(* PLC project tri_chain, Dassault Systèmes ControlBuild 2019 FD01 *)
(* stored: creationDateTime 2018-10-05T16:35:32-01:00 *)

CONFIGURATION tri_chain
  VAR_GLOBAL
    cp_trichain/ON AT 5 : BOOL := false;
    cp_trichain/run1 AT 6 : BOOL := false;
    cp_trichain/startSensor1 AT 7 : BOOL := false;
    cp_trichain/endSensor1 AT 8 : BOOL := false;
    cp_trichain/run2 AT 9 : BOOL := false;
    cp_trichain/startSensor2 AT 10 : BOOL := false;
    cp_trichain/endSensor2 AT 11 : BOOL := false;
    cp_trichain/run3 AT 12 : BOOL := false;
    cp_trichain/startSensor3 AT 13 : BOOL := false;
    cp_trichain/endSensor3 AT 14 : BOOL := false;
    cp_trichain/sensor1 AT 15 : BOOL := false;
    cp_trichain/sensor2 AT 16 : BOOL := false;
    cp_trichain/sensor3 AT 17 : BOOL := false;
    cp_trichain/endSensor AT 18 : BOOL := false;
    cp_trichain/endSensor4 AT 19 : BOOL := false;
    cp_trichain/mvt1 AT 20 : BOOL := false;
    cp_trichain/mvt2 AT 21 : BOOL := false;
    cp_trichain/mvt3 AT 22 : BOOL := false;
    cp_trichain/moveToLeft AT 24 : BOOL := false;
    cp_trichain/moveToRight AT 25 : BOOL := false;
    cp_trichain/chainMvt AT 26 : BOOL := false;
    cp_trichain/mvt4 AT 23 : BOOL := false;
    cp_trichain/chain1/globalRunning AT 5 : BOOL := false;
    cp_trichain/chain1/localRunning AT 6 : BOOL := false;
    cp_trichain/chain1/startSensor AT 7 : BOOL := false;
    cp_trichain/chain1/endSensor AT 8 : BOOL := false;
    cp_trichain/chain1/captureEnabled AT 27 : BOOL := false;
    cp_trichain/chain1/movement AT 20 : BOOL := false;
    cp_trichain/chain1/captureRequest AT 30 : BOOL := false;
    cp_trichain/chain1/captureFinished AT 31 : BOOL := false;
    cp_trichain/chain1/_X_10 AT 40 : BOOL := true;
    cp_trichain/chain1/_X_11 AT 41 : BOOL := false;
    cp_trichain/chain1/_X_12 AT 42 : BOOL := false;
    cp_trichain/chain1/_X_13 AT 43 : BOOL := false;
    cp_trichain/chain1/_X_14 AT 44 : BOOL := false;
    cp_trichain/chain1/_X_15 AT 45 : BOOL := false;
    cp_trichain/chain2/globalRunning AT 5 : BOOL := false;
    cp_trichain/chain2/localRunning AT 9 : BOOL := false;
    cp_trichain/chain2/startSensor AT 10 : BOOL := false;
    cp_trichain/chain2/endSensor AT 11 : BOOL := false;
    cp_trichain/chain2/captureEnabled AT 28 : BOOL := false;
    cp_trichain/chain2/movement AT 21 : BOOL := false;
    cp_trichain/chain2/captureRequest AT 32 : BOOL := false;
    cp_trichain/chain2/captureFinished AT 33 : BOOL := false;
    cp_trichain/chain2/_X_10 AT 50 : BOOL := true;
    cp_trichain/chain2/_X_11 AT 51 : BOOL := false;
    cp_trichain/chain2/_X_12 AT 52 : BOOL := false;
    cp_trichain/chain2/_X_13 AT 53 : BOOL := false;
    cp_trichain/chain2/_X_14 AT 54 : BOOL := false;
    cp_trichain/chain2/_X_15 AT 55 : BOOL := false;
    cp_trichain/chain3/globalRunning AT 5 : BOOL := false;
    cp_trichain/chain3/localRunning AT 12 : BOOL := false;
    cp_trichain/chain3/startSensor AT 13 : BOOL := false;
    cp_trichain/chain3/endSensor AT 14 : BOOL := false;
    cp_trichain/chain3/captureEnabled AT 29 : BOOL := false;
    cp_trichain/chain3/movement AT 22 : BOOL := false;
    cp_trichain/chain3/captureRequest AT 34 : BOOL := false;
    cp_trichain/chain3/captureFinished AT 35 : BOOL := false;
    cp_trichain/chain3/_X_10 AT 60 : BOOL := true;
    cp_trichain/chain3/_X_11 AT 61 : BOOL := false;
    cp_trichain/chain3/_X_12 AT 62 : BOOL := false;
    cp_trichain/chain3/_X_13 AT 63 : BOOL := false;
    cp_trichain/chain3/_X_14 AT 64 : BOOL := false;
    cp_trichain/chain3/_X_15 AT 65 : BOOL := false;
    cp_trichain/shuttleControl/globalRunning AT 5 : BOOL := false;
    cp_trichain/shuttleControl/sensorPos1 AT 15 : BOOL := false;
    cp_trichain/shuttleControl/sensorPos2 AT 16 : BOOL := false;
    cp_trichain/shuttleControl/sensorPos3 AT 17 : BOOL := false;
    cp_trichain/shuttleControl/requestCapture1 AT 30 : BOOL := false;
    cp_trichain/shuttleControl/endCapture1 AT 31 : BOOL := false;
    cp_trichain/shuttleControl/requestCapture2 AT 32 : BOOL := false;
    cp_trichain/shuttleControl/endCapture2 AT 33 : BOOL := false;
    cp_trichain/shuttleControl/requestCapture3 AT 34 : BOOL := false;
    cp_trichain/shuttleControl/endCapture3 AT 35 : BOOL := false;
    cp_trichain/shuttleControl/depositRequest AT 36 : BOOL := false;
    cp_trichain/shuttleControl/depositFinished AT 37 : BOOL := false;
    cp_trichain/shuttleControl/enableCapture1 AT 27 : BOOL := false;
    cp_trichain/shuttleControl/enableCapture2 AT 28 : BOOL := false;
    cp_trichain/shuttleControl/enableCapture3 AT 29 : BOOL := false;
    cp_trichain/shuttleControl/enableCapture AT 39 : BOOL := false;
    cp_trichain/shuttleControl/enableDeposit AT 38 : BOOL := false;
    cp_trichain/shuttleControl/moveToLeft AT 24 : BOOL := false;
    cp_trichain/shuttleControl/moveToRight AT 25 : BOOL := false;
    cp_trichain/shuttleControl/goTo1 AT 70 : BOOL := false;
    cp_trichain/shuttleControl/goTo2 AT 71 : BOOL := false;
    cp_trichain/shuttleControl/goTo3 AT 72 : BOOL := false;
    cp_trichain/shuttleControl/shuttleInPosition AT 73 : BOOL := false;
    cp_trichain/shuttleControl/_X_10 AT 74 : BOOL := true;
    cp_trichain/shuttleControl/_X_15 AT 82 : BOOL := false;
    cp_trichain/shuttleControl/_X_13 AT 80 : BOOL := false;
    cp_trichain/shuttleControl/_X_11 AT 75 : BOOL := false;
    cp_trichain/shuttleControl/_X_16 AT 83 : BOOL := false;
    cp_trichain/shuttleControl/_X_14 AT 81 : BOOL := false;
    cp_trichain/shuttleControl/_X_12 AT 76 : BOOL := false;
    cp_trichain/shuttleControl/_X_17 AT 77 : BOOL := false;
    cp_trichain/shuttleControl/_X_18 AT 78 : BOOL := false;
    cp_trichain/shuttleControl/_X_19 AT 79 : BOOL := false;
    cp_trichain/shuttleControl/_X_20 AT 84 : BOOL := true;
    cp_trichain/shuttleControl/_X_21 AT 85 : BOOL := false;
    cp_trichain/shuttleControl/_X_22 AT 86 : BOOL := false;
    cp_trichain/shuttleControl/_X_30 AT 87 : BOOL := true;
    cp_trichain/shuttleControl/_X_31 AT 88 : BOOL := false;
    cp_trichain/shuttleControl/_X_32 AT 89 : BOOL := false;
    cp_trichain/shuttleControl/_X_40 AT 90 : BOOL := true;
    cp_trichain/shuttleControl/_X_41 AT 91 : BOOL := false;
    cp_trichain/shuttleControl/_X_42 AT 92 : BOOL := false;
    cp_trichain/shuttleChain/globalRunning AT 5 : BOOL := false;
    cp_trichain/shuttleChain/endSensor AT 18 : BOOL := false;
    cp_trichain/shuttleChain/depositEnabled AT 38 : BOOL := false;
    cp_trichain/shuttleChain/captureEnabled AT 39 : BOOL := false;
    cp_trichain/shuttleChain/movement AT 26 : BOOL := false;
    cp_trichain/shuttleChain/depositRequest AT 36 : BOOL := false;
    cp_trichain/shuttleChain/depositFinished AT 37 : BOOL := false;
    cp_trichain/shuttleChain/_X_10 AT 108 : BOOL := true;
    cp_trichain/shuttleChain/_X_11 AT 109 : BOOL := false;
    cp_trichain/shuttleChain/_X_12 AT 110 : BOOL := false;
    cp_trichain/shuttleChain/_X_13 AT 111 : BOOL := false;
    cp_trichain/shuttleChain/_X_14 AT 112 : BOOL := false;
    cp_trichain/outputChain/globalRunning AT 5 : BOOL := false;
    cp_trichain/outputChain/depositEnabled AT 38 : BOOL := false;
    cp_trichain/outputChain/endSensor AT 19 : BOOL := false;
    cp_trichain/outputChain/movement AT 23 : BOOL := false;
    cp_trichain/outputChain/_X_10 AT 117 : BOOL := true;
    cp_trichain/outputChain/_X_11 AT 118 : BOOL := false;
    cp_trichain/outputChain/_X_12 AT 119 : BOOL := false;
    op_trichain/mvt1 AT 20 : BOOL := false;
    op_trichain/mvt2 AT 21 : BOOL := false;
    op_trichain/mvt3 AT 22 : BOOL := false;
    op_trichain/mvt4 AT 23 : BOOL := false;
    op_trichain/moveToLeft AT 24 : BOOL := false;
    op_trichain/moveToRight AT 25 : BOOL := false;
    op_trichain/chainMvt AT 26 : BOOL := false;
    op_trichain/ON AT 5 : BOOL := false;
    op_trichain/run1 AT 6 : BOOL := false;
    op_trichain/startSensor1 AT 7 : BOOL := false;
    op_trichain/endSensor1 AT 8 : BOOL := false;
    op_trichain/run2 AT 9 : BOOL := false;
    op_trichain/startSensor2 AT 10 : BOOL := false;
    op_trichain/endSensor2 AT 11 : BOOL := false;
    op_trichain/run3 AT 12 : BOOL := false;
    op_trichain/startSensor3 AT 13 : BOOL := false;
    op_trichain/endSensor3 AT 14 : BOOL := false;
    op_trichain/endSensor4 AT 19 : BOOL := false;
    op_trichain/sensor1 AT 15 : BOOL := false;
    op_trichain/sensor2 AT 16 : BOOL := false;
    op_trichain/sensor3 AT 17 : BOOL := false;
    op_trichain/endSensor AT 18 : BOOL := false;
    op_trichain/creation1/idProd AT 525 : DINT := 0;
    op_trichain/creation1/creationFailed AT 126 : BOOL := false;
    op_trichain/creation1/status_act_prod AT 526 : DINT := 0;
    op_trichain/creation1/m11 AT 17 : REAL := 1502.68;
    op_trichain/creation1/m12 AT 18 : REAL := 0.0;
    op_trichain/creation1/m13 AT 19 : REAL := -2.44921e-014;
    op_trichain/creation1/m14 AT 20 : REAL := 5480.36;
    op_trichain/creation1/m21 AT 21 : REAL := 0.0;
    op_trichain/creation1/m22 AT 22 : REAL := 2997.32;
    op_trichain/creation1/m23 AT 23 : REAL := 0.0;
    op_trichain/creation1/m24 AT 24 : REAL := 27006.2;
    op_trichain/creation1/m31 AT 25 : REAL := 3.68038e-013;
    op_trichain/creation1/m32 AT 26 : REAL := 0.0;
    op_trichain/creation1/m33 AT 27 : REAL := 100.0;
    op_trichain/creation1/m34 AT 28 : REAL := 1.0;
    op_trichain/creation1/m41 AT 29 : REAL := 0.0;
    op_trichain/creation1/m42 AT 30 : REAL := 0.0;
    op_trichain/creation1/m43 AT 31 : REAL := 0.0;
    op_trichain/creation1/m44 AT 32 : REAL := 1.0;
    op_trichain/creation1/px AT 33 : REAL := 5600.0;
    op_trichain/creation1/py AT 34 : REAL := 27000.0;
    op_trichain/creation1/pz AT 35 : REAL := 1.5;
    op_trichain/creation1/dx AT 36 : REAL := 1500.0;
    op_trichain/creation1/dy AT 37 : REAL := 3000.0;
    op_trichain/creation1/dz AT 38 : REAL := 100.0;
    op_trichain/creation1/presenceProduct AT 127 : BOOL := false;
    op_trichain/creation1/arrival_PB AT 128 : BOOL := false;
    op_trichain/creation1/time2reach AT 39 : REAL := 0.0;
    op_trichain/creation1/edge_arrival_PB AT 129 : BOOL := false;
    op_trichain/creation1/first AT 130 : BOOL := true;
    op_trichain/creation1/pulseType AT 131 : BOOL := true;
    op_trichain/creation1/pulseDuration AT 40 : REAL := 10.0;
    op_trichain/chain1/forward AT 20 : BOOL := false;
    op_trichain/chain1/localRun AT 6 : BOOL := false;
    op_trichain/chain1/start_sensor AT 7 : BOOL := false;
    op_trichain/chain1/end_sensor AT 8 : BOOL := false;
    op_trichain/chain1/motor1dir/forward AT 20 : BOOL := false;
    op_trichain/chain1/motor1dir/cmdSupply AT 138 : BOOL := true;
    op_trichain/chain1/motor1dir/sensorSupply AT 137 : BOOL := true;
    op_trichain/chain1/motor1dir/voltage380 AT 136 : BOOL := true;
    op_trichain/chain1/motor1dir/speedVal AT 42 : REAL := 0.0;
    op_trichain/chain1/motor1dir/speedPercent AT 41 : REAL := 0.0;
    op_trichain/chain1/motor1dir/thermal AT 135 : BOOL := false;
    op_trichain/chain1/motor1dir/forwardFB AT 134 : BOOL := false;
    op_trichain/chain1/motor1dir/increment AT 43 : REAL := 0.0;
    op_trichain/chain1/motor1dir/memoFwd AT 139 : BOOL := false;
    op_trichain/chain1/motor1dir/forwardState AT 140 : BOOL := false;
    op_trichain/chain1/motor1dir/wantedSpeed AT 44 : REAL := 0.0;
    op_trichain/chain1/motor1dir/nominalSpeed AT 45 : REAL := 500.0;
    op_trichain/chain1/motor1dir/nominalTime AT 46 : REAL := 0.1;
    op_trichain/chain1/motor1dir/thermalLogic AT 141 : BOOL := false;
    op_trichain/chain1/motor1dir/feedbackLogic AT 142 : BOOL := true;
    op_trichain/chain1/motor1dir/d_locking AT 143 : BOOL := false;
    op_trichain/chain1/motor1dir/v_d_locking AT 47 : REAL := 0.0;
    op_trichain/chain1/motor1dir/d_feedback AT 144 : BOOL := false;
    op_trichain/chain1/motor1dir/v_d_feedback AT 145 : BOOL := false;
    op_trichain/chain1/motor1dir/d_electrical AT 146 : BOOL := false;
    op_trichain/chain1/motor1dir/v_d_electrical AT 147 : BOOL := false;
    op_trichain/chain1/runButton/output AT 6 : BOOL := false;
    op_trichain/chain1/runButton/user_PushButton AT 148 : BOOL := false;
    op_trichain/chain1/runButton/time2reach AT 149 : BOOL := false;
    op_trichain/chain1/runButton/pulse_type AT 150 : BOOL := false;
    op_trichain/chain1/runButton/pulseDuration AT 48 : REAL := 2.0;
    op_trichain/chain1/start_sensor/sensorSupply AT 133 : BOOL := true;
    op_trichain/chain1/start_sensor/passing AT 7 : BOOL := false;
    op_trichain/chain1/start_sensor/status_act_prod AT 527 : DINT := 0;
    op_trichain/chain1/start_sensor/m11 AT 49 : REAL := 498.214;
    op_trichain/chain1/start_sensor/m12 AT 50 : REAL := 0.0;
    op_trichain/chain1/start_sensor/m13 AT 51 : REAL := -2.44921e-014;
    op_trichain/chain1/start_sensor/m14 AT 52 : REAL := 5223.22;
    op_trichain/chain1/start_sensor/m21 AT 53 : REAL := 0.0;
    op_trichain/chain1/start_sensor/m22 AT 54 : REAL := 498.214;
    op_trichain/chain1/start_sensor/m23 AT 55 : REAL := 0.0;
    op_trichain/chain1/start_sensor/m24 AT 56 : REAL := 26998.2;
    op_trichain/chain1/start_sensor/m31 AT 57 : REAL := 1.22023e-013;
    op_trichain/chain1/start_sensor/m32 AT 58 : REAL := 0.0;
    op_trichain/chain1/start_sensor/m33 AT 59 : REAL := 100.0;
    op_trichain/chain1/start_sensor/m34 AT 60 : REAL := 1.0;
    op_trichain/chain1/start_sensor/m41 AT 61 : REAL := 0.0;
    op_trichain/chain1/start_sensor/m42 AT 62 : REAL := 0.0;
    op_trichain/chain1/start_sensor/m43 AT 63 : REAL := 0.0;
    op_trichain/chain1/start_sensor/m44 AT 64 : REAL := 1.0;
    op_trichain/chain1/start_sensor/px AT 65 : REAL := 4500.0;
    op_trichain/chain1/start_sensor/py AT 66 : REAL := 27000.0;
    op_trichain/chain1/start_sensor/pz AT 67 : REAL := 0.0;
    op_trichain/chain1/start_sensor/dx AT 68 : REAL := 500.0;
    op_trichain/chain1/start_sensor/dy AT 69 : REAL := 500.0;
    op_trichain/chain1/start_sensor/dz AT 70 : REAL := 100.0;
    op_trichain/chain1/start_sensor/detection AT 151 : BOOL := false;
    op_trichain/chain1/start_sensor/passingLogic AT 152 : BOOL := true;
    op_trichain/chain1/start_sensor/d_passing AT 153 : BOOL := false;
    op_trichain/chain1/start_sensor/v_d_passing AT 154 : BOOL := true;
    op_trichain/chain1/end_sensor/sensorSupply AT 132 : BOOL := true;
    op_trichain/chain1/end_sensor/passing AT 8 : BOOL := false;
    op_trichain/chain1/end_sensor/status_act_prod AT 528 : DINT := 0;
    op_trichain/chain1/end_sensor/m11 AT 71 : REAL := 498.214;
    op_trichain/chain1/end_sensor/m12 AT 72 : REAL := 0.0;
    op_trichain/chain1/end_sensor/m13 AT 73 : REAL := -2.44921e-014;
    op_trichain/chain1/end_sensor/m14 AT 74 : REAL := 3334.82;
    op_trichain/chain1/end_sensor/m21 AT 75 : REAL := 0.0;
    op_trichain/chain1/end_sensor/m22 AT 76 : REAL := 498.214;
    op_trichain/chain1/end_sensor/m23 AT 77 : REAL := 0.0;
    op_trichain/chain1/end_sensor/m24 AT 78 : REAL := 19999.1;
    op_trichain/chain1/end_sensor/m31 AT 79 : REAL := 1.22023e-013;
    op_trichain/chain1/end_sensor/m32 AT 80 : REAL := 0.0;
    op_trichain/chain1/end_sensor/m33 AT 81 : REAL := 100.0;
    op_trichain/chain1/end_sensor/m34 AT 82 : REAL := 1.05;
    op_trichain/chain1/end_sensor/m41 AT 83 : REAL := 0.0;
    op_trichain/chain1/end_sensor/m42 AT 84 : REAL := 0.0;
    op_trichain/chain1/end_sensor/m43 AT 85 : REAL := 0.0;
    op_trichain/chain1/end_sensor/m44 AT 86 : REAL := 1.0;
    op_trichain/chain1/end_sensor/px AT 87 : REAL := 2850.0;
    op_trichain/chain1/end_sensor/py AT 88 : REAL := 20000.0;
    op_trichain/chain1/end_sensor/pz AT 89 : REAL := 0.0;
    op_trichain/chain1/end_sensor/dx AT 90 : REAL := 500.0;
    op_trichain/chain1/end_sensor/dy AT 91 : REAL := 500.0;
    op_trichain/chain1/end_sensor/dz AT 92 : REAL := 100.0;
    op_trichain/chain1/end_sensor/detection AT 155 : BOOL := false;
    op_trichain/chain1/end_sensor/passingLogic AT 156 : BOOL := true;
    op_trichain/chain1/end_sensor/d_passing AT 157 : BOOL := false;
    op_trichain/chain1/end_sensor/v_d_passing AT 158 : BOOL := true;
    op_trichain/chain1/chain/linearSpeed AT 42 : REAL := 0.0;
    op_trichain/chain1/chain/status_act_prod AT 529 : DINT := 0;
    op_trichain/chain1/chain/m11 AT 93 : REAL := 4001.79;
    op_trichain/chain1/chain/m12 AT 94 : REAL := 0.0;
    op_trichain/chain1/chain/m13 AT 95 : REAL := -2.44921e-014;
    op_trichain/chain1/chain/m14 AT 96 : REAL := 2981.25;
    op_trichain/chain1/chain/m21 AT 97 : REAL := 0.0;
    op_trichain/chain1/chain/m22 AT 98 : REAL := 9996.43;
    op_trichain/chain1/chain/m23 AT 99 : REAL := 0.0;
    op_trichain/chain1/chain/m24 AT 100 : REAL := 18102.7;
    op_trichain/chain1/chain/m31 AT 101 : REAL := 9.80123e-013;
    op_trichain/chain1/chain/m32 AT 102 : REAL := 0.0;
    op_trichain/chain1/chain/m33 AT 103 : REAL := 100.0;
    op_trichain/chain1/chain/m34 AT 104 : REAL := 1.0;
    op_trichain/chain1/chain/m41 AT 105 : REAL := 0.0;
    op_trichain/chain1/chain/m42 AT 106 : REAL := 0.0;
    op_trichain/chain1/chain/m43 AT 107 : REAL := 0.0;
    op_trichain/chain1/chain/m44 AT 108 : REAL := 1.0;
    op_trichain/chain1/chain/px AT 109 : REAL := 2500.0;
    op_trichain/chain1/chain/py AT 110 : REAL := 18100.0;
    op_trichain/chain1/chain/pz AT 111 : REAL := 1.0;
    op_trichain/chain1/chain/dx AT 112 : REAL := 4000.0;
    op_trichain/chain1/chain/dy AT 113 : REAL := 10000.0;
    op_trichain/chain1/chain/dz AT 114 : REAL := 100.0;
    op_trichain/chain1/chain/sProduct AT 115 : REAL := 0.0;
    op_trichain/chain1/chain/interaction AT 159 : BOOL := false;
    op_trichain/chain1/chain/d_locking AT 160 : BOOL := false;
    op_trichain/chain1/chain/v_d_locking AT 161 : BOOL := false;
    op_trichain/chain2/forward AT 21 : BOOL := false;
    op_trichain/chain2/localRun AT 9 : BOOL := false;
    op_trichain/chain2/start_sensor AT 10 : BOOL := false;
    op_trichain/chain2/end_sensor AT 11 : BOOL := false;
    op_trichain/chain2/motor1dir/forward AT 21 : BOOL := false;
    op_trichain/chain2/motor1dir/cmdSupply AT 168 : BOOL := true;
    op_trichain/chain2/motor1dir/sensorSupply AT 167 : BOOL := true;
    op_trichain/chain2/motor1dir/voltage380 AT 166 : BOOL := true;
    op_trichain/chain2/motor1dir/speedVal AT 117 : REAL := 0.0;
    op_trichain/chain2/motor1dir/speedPercent AT 116 : REAL := 0.0;
    op_trichain/chain2/motor1dir/thermal AT 165 : BOOL := false;
    op_trichain/chain2/motor1dir/forwardFB AT 164 : BOOL := false;
    op_trichain/chain2/motor1dir/increment AT 118 : REAL := 0.0;
    op_trichain/chain2/motor1dir/memoFwd AT 169 : BOOL := false;
    op_trichain/chain2/motor1dir/forwardState AT 170 : BOOL := false;
    op_trichain/chain2/motor1dir/wantedSpeed AT 119 : REAL := 0.0;
    op_trichain/chain2/motor1dir/nominalSpeed AT 120 : REAL := 500.0;
    op_trichain/chain2/motor1dir/nominalTime AT 121 : REAL := 0.1;
    op_trichain/chain2/motor1dir/thermalLogic AT 171 : BOOL := false;
    op_trichain/chain2/motor1dir/feedbackLogic AT 172 : BOOL := true;
    op_trichain/chain2/motor1dir/d_locking AT 173 : BOOL := false;
    op_trichain/chain2/motor1dir/v_d_locking AT 122 : REAL := 0.0;
    op_trichain/chain2/motor1dir/d_feedback AT 174 : BOOL := false;
    op_trichain/chain2/motor1dir/v_d_feedback AT 175 : BOOL := false;
    op_trichain/chain2/motor1dir/d_electrical AT 176 : BOOL := false;
    op_trichain/chain2/motor1dir/v_d_electrical AT 177 : BOOL := false;
    op_trichain/chain2/runButton/output AT 9 : BOOL := false;
    op_trichain/chain2/runButton/user_PushButton AT 178 : BOOL := false;
    op_trichain/chain2/runButton/time2reach AT 179 : BOOL := false;
    op_trichain/chain2/runButton/pulse_type AT 180 : BOOL := false;
    op_trichain/chain2/runButton/pulseDuration AT 123 : REAL := 2.0;
    op_trichain/chain2/start_sensor/sensorSupply AT 163 : BOOL := true;
    op_trichain/chain2/start_sensor/passing AT 10 : BOOL := false;
    op_trichain/chain2/start_sensor/status_act_prod AT 530 : DINT := 0;
    op_trichain/chain2/start_sensor/m11 AT 124 : REAL := 500.0;
    op_trichain/chain2/start_sensor/m12 AT 125 : REAL := 0.0;
    op_trichain/chain2/start_sensor/m13 AT 126 : REAL := 0.0;
    op_trichain/chain2/start_sensor/m14 AT 127 : REAL := 8500.0;
    op_trichain/chain2/start_sensor/m21 AT 128 : REAL := 0.0;
    op_trichain/chain2/start_sensor/m22 AT 129 : REAL := 500.0;
    op_trichain/chain2/start_sensor/m23 AT 130 : REAL := 0.0;
    op_trichain/chain2/start_sensor/m24 AT 131 : REAL := 27000.0;
    op_trichain/chain2/start_sensor/m31 AT 132 : REAL := 0.0;
    op_trichain/chain2/start_sensor/m32 AT 133 : REAL := 0.0;
    op_trichain/chain2/start_sensor/m33 AT 134 : REAL := 100.0;
    op_trichain/chain2/start_sensor/m34 AT 135 : REAL := 0.0;
    op_trichain/chain2/start_sensor/m41 AT 136 : REAL := 0.0;
    op_trichain/chain2/start_sensor/m42 AT 137 : REAL := 0.0;
    op_trichain/chain2/start_sensor/m43 AT 138 : REAL := 0.0;
    op_trichain/chain2/start_sensor/m44 AT 139 : REAL := 1.0;
    op_trichain/chain2/start_sensor/px AT 140 : REAL := 8500.0;
    op_trichain/chain2/start_sensor/py AT 141 : REAL := 27000.0;
    op_trichain/chain2/start_sensor/pz AT 142 : REAL := 0.0;
    op_trichain/chain2/start_sensor/dx AT 143 : REAL := 500.0;
    op_trichain/chain2/start_sensor/dy AT 144 : REAL := 500.0;
    op_trichain/chain2/start_sensor/dz AT 145 : REAL := 100.0;
    op_trichain/chain2/start_sensor/detection AT 181 : BOOL := false;
    op_trichain/chain2/start_sensor/passingLogic AT 182 : BOOL := true;
    op_trichain/chain2/start_sensor/d_passing AT 183 : BOOL := false;
    op_trichain/chain2/start_sensor/v_d_passing AT 184 : BOOL := true;
    op_trichain/chain2/end_sensor/sensorSupply AT 162 : BOOL := true;
    op_trichain/chain2/end_sensor/passing AT 11 : BOOL := false;
    op_trichain/chain2/end_sensor/status_act_prod AT 531 : DINT := 0;
    op_trichain/chain2/end_sensor/m11 AT 146 : REAL := 500.0;
    op_trichain/chain2/end_sensor/m12 AT 147 : REAL := 0.0;
    op_trichain/chain2/end_sensor/m13 AT 148 : REAL := 0.0;
    op_trichain/chain2/end_sensor/m14 AT 149 : REAL := 6900.0;
    op_trichain/chain2/end_sensor/m21 AT 150 : REAL := 0.0;
    op_trichain/chain2/end_sensor/m22 AT 151 : REAL := 500.0;
    op_trichain/chain2/end_sensor/m23 AT 152 : REAL := 0.0;
    op_trichain/chain2/end_sensor/m24 AT 153 : REAL := 20000.0;
    op_trichain/chain2/end_sensor/m31 AT 154 : REAL := 0.0;
    op_trichain/chain2/end_sensor/m32 AT 155 : REAL := 0.0;
    op_trichain/chain2/end_sensor/m33 AT 156 : REAL := 100.0;
    op_trichain/chain2/end_sensor/m34 AT 157 : REAL := 0.0;
    op_trichain/chain2/end_sensor/m41 AT 158 : REAL := 0.0;
    op_trichain/chain2/end_sensor/m42 AT 159 : REAL := 0.0;
    op_trichain/chain2/end_sensor/m43 AT 160 : REAL := 0.0;
    op_trichain/chain2/end_sensor/m44 AT 161 : REAL := 1.0;
    op_trichain/chain2/end_sensor/px AT 162 : REAL := 6900.0;
    op_trichain/chain2/end_sensor/py AT 163 : REAL := 20000.0;
    op_trichain/chain2/end_sensor/pz AT 164 : REAL := 0.0;
    op_trichain/chain2/end_sensor/dx AT 165 : REAL := 500.0;
    op_trichain/chain2/end_sensor/dy AT 166 : REAL := 500.0;
    op_trichain/chain2/end_sensor/dz AT 167 : REAL := 100.0;
    op_trichain/chain2/end_sensor/detection AT 185 : BOOL := false;
    op_trichain/chain2/end_sensor/passingLogic AT 186 : BOOL := true;
    op_trichain/chain2/end_sensor/d_passing AT 187 : BOOL := false;
    op_trichain/chain2/end_sensor/v_d_passing AT 188 : BOOL := true;
    op_trichain/chain2/chain/linearSpeed AT 117 : REAL := 0.0;
    op_trichain/chain2/chain/status_act_prod AT 532 : DINT := 0;
    op_trichain/chain2/chain/m11 AT 168 : REAL := 4000.0;
    op_trichain/chain2/chain/m12 AT 169 : REAL := 0.0;
    op_trichain/chain2/chain/m13 AT 170 : REAL := 0.0;
    op_trichain/chain2/chain/m14 AT 171 : REAL := 6500.0;
    op_trichain/chain2/chain/m21 AT 172 : REAL := 0.0;
    op_trichain/chain2/chain/m22 AT 173 : REAL := 10000.0;
    op_trichain/chain2/chain/m23 AT 174 : REAL := 0.0;
    op_trichain/chain2/chain/m24 AT 175 : REAL := 18100.0;
    op_trichain/chain2/chain/m31 AT 176 : REAL := 0.0;
    op_trichain/chain2/chain/m32 AT 177 : REAL := 0.0;
    op_trichain/chain2/chain/m33 AT 178 : REAL := 100.0;
    op_trichain/chain2/chain/m34 AT 179 : REAL := 0.0;
    op_trichain/chain2/chain/m41 AT 180 : REAL := 0.0;
    op_trichain/chain2/chain/m42 AT 181 : REAL := 0.0;
    op_trichain/chain2/chain/m43 AT 182 : REAL := 0.0;
    op_trichain/chain2/chain/m44 AT 183 : REAL := 1.0;
    op_trichain/chain2/chain/px AT 184 : REAL := 6500.0;
    op_trichain/chain2/chain/py AT 185 : REAL := 18100.0;
    op_trichain/chain2/chain/pz AT 186 : REAL := 0.0;
    op_trichain/chain2/chain/dx AT 187 : REAL := 4000.0;
    op_trichain/chain2/chain/dy AT 188 : REAL := 10000.0;
    op_trichain/chain2/chain/dz AT 189 : REAL := 100.0;
    op_trichain/chain2/chain/sProduct AT 190 : REAL := 0.0;
    op_trichain/chain2/chain/interaction AT 189 : BOOL := false;
    op_trichain/chain2/chain/d_locking AT 190 : BOOL := false;
    op_trichain/chain2/chain/v_d_locking AT 191 : BOOL := false;
    op_trichain/creation2/idProd AT 524 : DINT := 0;
    op_trichain/creation2/creationFailed AT 125 : BOOL := false;
    op_trichain/creation2/status_act_prod AT 533 : DINT := 0;
    op_trichain/creation2/m11 AT 191 : REAL := 1500.0;
    op_trichain/creation2/m12 AT 192 : REAL := 0.0;
    op_trichain/creation2/m13 AT 193 : REAL := 0.0;
    op_trichain/creation2/m14 AT 194 : REAL := 9000.0;
    op_trichain/creation2/m21 AT 195 : REAL := 0.0;
    op_trichain/creation2/m22 AT 196 : REAL := 3000.0;
    op_trichain/creation2/m23 AT 197 : REAL := 0.0;
    op_trichain/creation2/m24 AT 198 : REAL := 27000.0;
    op_trichain/creation2/m31 AT 199 : REAL := 0.0;
    op_trichain/creation2/m32 AT 200 : REAL := 0.0;
    op_trichain/creation2/m33 AT 201 : REAL := 100.0;
    op_trichain/creation2/m34 AT 202 : REAL := 0.0;
    op_trichain/creation2/m41 AT 203 : REAL := 0.0;
    op_trichain/creation2/m42 AT 204 : REAL := 0.0;
    op_trichain/creation2/m43 AT 205 : REAL := 0.0;
    op_trichain/creation2/m44 AT 206 : REAL := 1.0;
    op_trichain/creation2/px AT 207 : REAL := 8990.0;
    op_trichain/creation2/py AT 208 : REAL := 27000.0;
    op_trichain/creation2/pz AT 209 : REAL := 1.5;
    op_trichain/creation2/dx AT 210 : REAL := 1500.0;
    op_trichain/creation2/dy AT 211 : REAL := 3000.0;
    op_trichain/creation2/dz AT 212 : REAL := 100.0;
    op_trichain/creation2/presenceProduct AT 192 : BOOL := false;
    op_trichain/creation2/arrival_PB AT 193 : BOOL := false;
    op_trichain/creation2/time2reach AT 213 : REAL := 0.0;
    op_trichain/creation2/edge_arrival_PB AT 194 : BOOL := false;
    op_trichain/creation2/first AT 195 : BOOL := true;
    op_trichain/creation2/pulseType AT 196 : BOOL := true;
    op_trichain/creation2/pulseDuration AT 214 : REAL := 10.0;
    op_trichain/chain3/forward AT 22 : BOOL := false;
    op_trichain/chain3/localRun AT 12 : BOOL := false;
    op_trichain/chain3/start_sensor AT 13 : BOOL := false;
    op_trichain/chain3/end_sensor AT 14 : BOOL := false;
    op_trichain/chain3/motor1dir/forward AT 22 : BOOL := false;
    op_trichain/chain3/motor1dir/cmdSupply AT 203 : BOOL := true;
    op_trichain/chain3/motor1dir/sensorSupply AT 202 : BOOL := true;
    op_trichain/chain3/motor1dir/voltage380 AT 201 : BOOL := true;
    op_trichain/chain3/motor1dir/speedVal AT 216 : REAL := 0.0;
    op_trichain/chain3/motor1dir/speedPercent AT 215 : REAL := 0.0;
    op_trichain/chain3/motor1dir/thermal AT 200 : BOOL := false;
    op_trichain/chain3/motor1dir/forwardFB AT 199 : BOOL := false;
    op_trichain/chain3/motor1dir/increment AT 217 : REAL := 0.0;
    op_trichain/chain3/motor1dir/memoFwd AT 204 : BOOL := false;
    op_trichain/chain3/motor1dir/forwardState AT 205 : BOOL := false;
    op_trichain/chain3/motor1dir/wantedSpeed AT 218 : REAL := 0.0;
    op_trichain/chain3/motor1dir/nominalSpeed AT 219 : REAL := 500.0;
    op_trichain/chain3/motor1dir/nominalTime AT 220 : REAL := 0.1;
    op_trichain/chain3/motor1dir/thermalLogic AT 206 : BOOL := false;
    op_trichain/chain3/motor1dir/feedbackLogic AT 207 : BOOL := true;
    op_trichain/chain3/motor1dir/d_locking AT 208 : BOOL := false;
    op_trichain/chain3/motor1dir/v_d_locking AT 221 : REAL := 0.0;
    op_trichain/chain3/motor1dir/d_feedback AT 209 : BOOL := false;
    op_trichain/chain3/motor1dir/v_d_feedback AT 210 : BOOL := false;
    op_trichain/chain3/motor1dir/d_electrical AT 211 : BOOL := false;
    op_trichain/chain3/motor1dir/v_d_electrical AT 212 : BOOL := false;
    op_trichain/chain3/runButton/output AT 12 : BOOL := false;
    op_trichain/chain3/runButton/user_PushButton AT 213 : BOOL := false;
    op_trichain/chain3/runButton/time2reach AT 214 : BOOL := false;
    op_trichain/chain3/runButton/pulse_type AT 215 : BOOL := false;
    op_trichain/chain3/runButton/pulseDuration AT 222 : REAL := 2.0;
    op_trichain/chain3/start_sensor/sensorSupply AT 198 : BOOL := true;
    op_trichain/chain3/start_sensor/passing AT 13 : BOOL := false;
    op_trichain/chain3/start_sensor/status_act_prod AT 534 : DINT := 0;
    op_trichain/chain3/start_sensor/m11 AT 223 : REAL := 500.0;
    op_trichain/chain3/start_sensor/m12 AT 224 : REAL := 0.0;
    op_trichain/chain3/start_sensor/m13 AT 225 : REAL := 0.0;
    op_trichain/chain3/start_sensor/m14 AT 226 : REAL := 12500.0;
    op_trichain/chain3/start_sensor/m21 AT 227 : REAL := 0.0;
    op_trichain/chain3/start_sensor/m22 AT 228 : REAL := 500.0;
    op_trichain/chain3/start_sensor/m23 AT 229 : REAL := 0.0;
    op_trichain/chain3/start_sensor/m24 AT 230 : REAL := 27000.0;
    op_trichain/chain3/start_sensor/m31 AT 231 : REAL := 0.0;
    op_trichain/chain3/start_sensor/m32 AT 232 : REAL := 0.0;
    op_trichain/chain3/start_sensor/m33 AT 233 : REAL := 100.0;
    op_trichain/chain3/start_sensor/m34 AT 234 : REAL := 0.0;
    op_trichain/chain3/start_sensor/m41 AT 235 : REAL := 0.0;
    op_trichain/chain3/start_sensor/m42 AT 236 : REAL := 0.0;
    op_trichain/chain3/start_sensor/m43 AT 237 : REAL := 0.0;
    op_trichain/chain3/start_sensor/m44 AT 238 : REAL := 1.0;
    op_trichain/chain3/start_sensor/px AT 239 : REAL := 12500.0;
    op_trichain/chain3/start_sensor/py AT 240 : REAL := 27000.0;
    op_trichain/chain3/start_sensor/pz AT 241 : REAL := 0.0;
    op_trichain/chain3/start_sensor/dx AT 242 : REAL := 500.0;
    op_trichain/chain3/start_sensor/dy AT 243 : REAL := 500.0;
    op_trichain/chain3/start_sensor/dz AT 244 : REAL := 100.0;
    op_trichain/chain3/start_sensor/detection AT 216 : BOOL := false;
    op_trichain/chain3/start_sensor/passingLogic AT 217 : BOOL := true;
    op_trichain/chain3/start_sensor/d_passing AT 218 : BOOL := false;
    op_trichain/chain3/start_sensor/v_d_passing AT 219 : BOOL := true;
    op_trichain/chain3/end_sensor/sensorSupply AT 197 : BOOL := true;
    op_trichain/chain3/end_sensor/passing AT 14 : BOOL := false;
    op_trichain/chain3/end_sensor/status_act_prod AT 535 : DINT := 0;
    op_trichain/chain3/end_sensor/m11 AT 245 : REAL := 500.0;
    op_trichain/chain3/end_sensor/m12 AT 246 : REAL := 0.0;
    op_trichain/chain3/end_sensor/m13 AT 247 : REAL := 0.0;
    op_trichain/chain3/end_sensor/m14 AT 248 : REAL := 10950.0;
    op_trichain/chain3/end_sensor/m21 AT 249 : REAL := 0.0;
    op_trichain/chain3/end_sensor/m22 AT 250 : REAL := 500.0;
    op_trichain/chain3/end_sensor/m23 AT 251 : REAL := 0.0;
    op_trichain/chain3/end_sensor/m24 AT 252 : REAL := 20000.0;
    op_trichain/chain3/end_sensor/m31 AT 253 : REAL := 0.0;
    op_trichain/chain3/end_sensor/m32 AT 254 : REAL := 0.0;
    op_trichain/chain3/end_sensor/m33 AT 255 : REAL := 100.0;
    op_trichain/chain3/end_sensor/m34 AT 256 : REAL := 0.0;
    op_trichain/chain3/end_sensor/m41 AT 257 : REAL := 0.0;
    op_trichain/chain3/end_sensor/m42 AT 258 : REAL := 0.0;
    op_trichain/chain3/end_sensor/m43 AT 259 : REAL := 0.0;
    op_trichain/chain3/end_sensor/m44 AT 260 : REAL := 1.0;
    op_trichain/chain3/end_sensor/px AT 261 : REAL := 10950.0;
    op_trichain/chain3/end_sensor/py AT 262 : REAL := 20000.0;
    op_trichain/chain3/end_sensor/pz AT 263 : REAL := 0.0;
    op_trichain/chain3/end_sensor/dx AT 264 : REAL := 0.0;
    op_trichain/chain3/end_sensor/dy AT 265 : REAL := 0.0;
    op_trichain/chain3/end_sensor/dz AT 266 : REAL := 0.0;
    op_trichain/chain3/end_sensor/detection AT 220 : BOOL := false;
    op_trichain/chain3/end_sensor/passingLogic AT 221 : BOOL := true;
    op_trichain/chain3/end_sensor/d_passing AT 222 : BOOL := false;
    op_trichain/chain3/end_sensor/v_d_passing AT 223 : BOOL := true;
    op_trichain/chain3/chain/linearSpeed AT 216 : REAL := 0.0;
    op_trichain/chain3/chain/status_act_prod AT 536 : DINT := 0;
    op_trichain/chain3/chain/m11 AT 267 : REAL := 4000.0;
    op_trichain/chain3/chain/m12 AT 268 : REAL := 0.0;
    op_trichain/chain3/chain/m13 AT 269 : REAL := 0.0;
    op_trichain/chain3/chain/m14 AT 270 : REAL := 10500.0;
    op_trichain/chain3/chain/m21 AT 271 : REAL := 0.0;
    op_trichain/chain3/chain/m22 AT 272 : REAL := 10000.0;
    op_trichain/chain3/chain/m23 AT 273 : REAL := 0.0;
    op_trichain/chain3/chain/m24 AT 274 : REAL := 18100.0;
    op_trichain/chain3/chain/m31 AT 275 : REAL := 0.0;
    op_trichain/chain3/chain/m32 AT 276 : REAL := 0.0;
    op_trichain/chain3/chain/m33 AT 277 : REAL := 100.0;
    op_trichain/chain3/chain/m34 AT 278 : REAL := 0.0;
    op_trichain/chain3/chain/m41 AT 279 : REAL := 0.0;
    op_trichain/chain3/chain/m42 AT 280 : REAL := 0.0;
    op_trichain/chain3/chain/m43 AT 281 : REAL := 0.0;
    op_trichain/chain3/chain/m44 AT 282 : REAL := 1.0;
    op_trichain/chain3/chain/px AT 283 : REAL := 10500.0;
    op_trichain/chain3/chain/py AT 284 : REAL := 18100.0;
    op_trichain/chain3/chain/pz AT 285 : REAL := 0.0;
    op_trichain/chain3/chain/dx AT 286 : REAL := 4000.0;
    op_trichain/chain3/chain/dy AT 287 : REAL := 10000.0;
    op_trichain/chain3/chain/dz AT 288 : REAL := 100.0;
    op_trichain/chain3/chain/sProduct AT 289 : REAL := 0.0;
    op_trichain/chain3/chain/interaction AT 224 : BOOL := false;
    op_trichain/chain3/chain/d_locking AT 225 : BOOL := false;
    op_trichain/chain3/chain/v_d_locking AT 226 : BOOL := false;
    op_trichain/outputChain/forward AT 23 : BOOL := false;
    op_trichain/outputChain/localRun AT 124 : BOOL := false;
    op_trichain/outputChain/start_sensor AT 123 : BOOL := false;
    op_trichain/outputChain/end_sensor AT 19 : BOOL := false;
    op_trichain/outputChain/motor1dir/forward AT 23 : BOOL := false;
    op_trichain/outputChain/motor1dir/cmdSupply AT 233 : BOOL := true;
    op_trichain/outputChain/motor1dir/sensorSupply AT 232 : BOOL := true;
    op_trichain/outputChain/motor1dir/voltage380 AT 231 : BOOL := true;
    op_trichain/outputChain/motor1dir/speedVal AT 291 : REAL := 0.0;
    op_trichain/outputChain/motor1dir/speedPercent AT 290 : REAL := 0.0;
    op_trichain/outputChain/motor1dir/thermal AT 230 : BOOL := false;
    op_trichain/outputChain/motor1dir/forwardFB AT 229 : BOOL := false;
    op_trichain/outputChain/motor1dir/increment AT 292 : REAL := 0.0;
    op_trichain/outputChain/motor1dir/memoFwd AT 234 : BOOL := false;
    op_trichain/outputChain/motor1dir/forwardState AT 235 : BOOL := false;
    op_trichain/outputChain/motor1dir/wantedSpeed AT 293 : REAL := 0.0;
    op_trichain/outputChain/motor1dir/nominalSpeed AT 294 : REAL := 500.0;
    op_trichain/outputChain/motor1dir/nominalTime AT 295 : REAL := 0.1;
    op_trichain/outputChain/motor1dir/thermalLogic AT 236 : BOOL := false;
    op_trichain/outputChain/motor1dir/feedbackLogic AT 237 : BOOL := true;
    op_trichain/outputChain/motor1dir/d_locking AT 238 : BOOL := false;
    op_trichain/outputChain/motor1dir/v_d_locking AT 296 : REAL := 0.0;
    op_trichain/outputChain/motor1dir/d_feedback AT 239 : BOOL := false;
    op_trichain/outputChain/motor1dir/v_d_feedback AT 240 : BOOL := false;
    op_trichain/outputChain/motor1dir/d_electrical AT 241 : BOOL := false;
    op_trichain/outputChain/motor1dir/v_d_electrical AT 242 : BOOL := false;
    op_trichain/outputChain/runButton/output AT 124 : BOOL := false;
    op_trichain/outputChain/runButton/user_PushButton AT 243 : BOOL := false;
    op_trichain/outputChain/runButton/time2reach AT 244 : BOOL := false;
    op_trichain/outputChain/runButton/pulse_type AT 245 : BOOL := false;
    op_trichain/outputChain/runButton/pulseDuration AT 297 : REAL := 2.0;
    op_trichain/outputChain/start_sensor/sensorSupply AT 228 : BOOL := true;
    op_trichain/outputChain/start_sensor/passing AT 123 : BOOL := false;
    op_trichain/outputChain/start_sensor/status_act_prod AT 537 : DINT := 0;
    op_trichain/outputChain/start_sensor/m11 AT 298 : REAL := 498.214;
    op_trichain/outputChain/start_sensor/m12 AT 299 : REAL := 0.0;
    op_trichain/outputChain/start_sensor/m13 AT 300 : REAL := 0.0;
    op_trichain/outputChain/start_sensor/m14 AT 301 : REAL := 9675.0;
    op_trichain/outputChain/start_sensor/m21 AT 302 : REAL := 0.0;
    op_trichain/outputChain/start_sensor/m22 AT 303 : REAL := 498.214;
    op_trichain/outputChain/start_sensor/m23 AT 304 : REAL := 0.0;
    op_trichain/outputChain/start_sensor/m24 AT 305 : REAL := 11987.5;
    op_trichain/outputChain/start_sensor/m31 AT 306 : REAL := 0.0;
    op_trichain/outputChain/start_sensor/m32 AT 307 : REAL := 0.0;
    op_trichain/outputChain/start_sensor/m33 AT 308 : REAL := 100.0;
    op_trichain/outputChain/start_sensor/m34 AT 309 : REAL := 1.06;
    op_trichain/outputChain/start_sensor/m41 AT 310 : REAL := 0.0;
    op_trichain/outputChain/start_sensor/m42 AT 311 : REAL := 0.0;
    op_trichain/outputChain/start_sensor/m43 AT 312 : REAL := 0.0;
    op_trichain/outputChain/start_sensor/m44 AT 313 : REAL := 1.0;
    op_trichain/outputChain/start_sensor/px AT 314 : REAL := 0.0;
    op_trichain/outputChain/start_sensor/py AT 315 : REAL := 0.0;
    op_trichain/outputChain/start_sensor/pz AT 316 : REAL := 0.0;
    op_trichain/outputChain/start_sensor/dx AT 317 : REAL := 500.0;
    op_trichain/outputChain/start_sensor/dy AT 318 : REAL := 500.0;
    op_trichain/outputChain/start_sensor/dz AT 319 : REAL := 100.0;
    op_trichain/outputChain/start_sensor/detection AT 246 : BOOL := false;
    op_trichain/outputChain/start_sensor/passingLogic AT 247 : BOOL := true;
    op_trichain/outputChain/start_sensor/d_passing AT 248 : BOOL := false;
    op_trichain/outputChain/start_sensor/v_d_passing AT 249 : BOOL := true;
    op_trichain/outputChain/end_sensor/sensorSupply AT 227 : BOOL := true;
    op_trichain/outputChain/end_sensor/passing AT 19 : BOOL := false;
    op_trichain/outputChain/end_sensor/status_act_prod AT 538 : DINT := 0;
    op_trichain/outputChain/end_sensor/m11 AT 320 : REAL := 500.0;
    op_trichain/outputChain/end_sensor/m12 AT 321 : REAL := 0.0;
    op_trichain/outputChain/end_sensor/m13 AT 322 : REAL := 0.0;
    op_trichain/outputChain/end_sensor/m14 AT 323 : REAL := 7450.0;
    op_trichain/outputChain/end_sensor/m21 AT 324 : REAL := 0.0;
    op_trichain/outputChain/end_sensor/m22 AT 325 : REAL := 500.0;
    op_trichain/outputChain/end_sensor/m23 AT 326 : REAL := 0.0;
    op_trichain/outputChain/end_sensor/m24 AT 327 : REAL := 4800.0;
    op_trichain/outputChain/end_sensor/m31 AT 328 : REAL := 0.0;
    op_trichain/outputChain/end_sensor/m32 AT 329 : REAL := 0.0;
    op_trichain/outputChain/end_sensor/m33 AT 330 : REAL := 100.0;
    op_trichain/outputChain/end_sensor/m34 AT 331 : REAL := 1.0;
    op_trichain/outputChain/end_sensor/m41 AT 332 : REAL := 0.0;
    op_trichain/outputChain/end_sensor/m42 AT 333 : REAL := 0.0;
    op_trichain/outputChain/end_sensor/m43 AT 334 : REAL := 0.0;
    op_trichain/outputChain/end_sensor/m44 AT 335 : REAL := 1.0;
    op_trichain/outputChain/end_sensor/px AT 336 : REAL := 7450.0;
    op_trichain/outputChain/end_sensor/py AT 337 : REAL := 4800.0;
    op_trichain/outputChain/end_sensor/pz AT 338 : REAL := 0.0;
    op_trichain/outputChain/end_sensor/dx AT 339 : REAL := 500.0;
    op_trichain/outputChain/end_sensor/dy AT 340 : REAL := 500.0;
    op_trichain/outputChain/end_sensor/dz AT 341 : REAL := 100.0;
    op_trichain/outputChain/end_sensor/detection AT 250 : BOOL := false;
    op_trichain/outputChain/end_sensor/passingLogic AT 251 : BOOL := true;
    op_trichain/outputChain/end_sensor/d_passing AT 252 : BOOL := false;
    op_trichain/outputChain/end_sensor/v_d_passing AT 253 : BOOL := true;
    op_trichain/outputChain/chain/linearSpeed AT 291 : REAL := 0.0;
    op_trichain/outputChain/chain/status_act_prod AT 539 : DINT := 0;
    op_trichain/outputChain/chain/m11 AT 342 : REAL := 4001.79;
    op_trichain/outputChain/chain/m12 AT 343 : REAL := 0.0;
    op_trichain/outputChain/chain/m13 AT 344 : REAL := 0.0;
    op_trichain/outputChain/chain/m14 AT 345 : REAL := 7003.57;
    op_trichain/outputChain/chain/m21 AT 346 : REAL := 0.0;
    op_trichain/outputChain/chain/m22 AT 347 : REAL := 9996.43;
    op_trichain/outputChain/chain/m23 AT 348 : REAL := 0.0;
    op_trichain/outputChain/chain/m24 AT 349 : REAL := 2352.06;
    op_trichain/outputChain/chain/m31 AT 350 : REAL := 0.0;
    op_trichain/outputChain/chain/m32 AT 351 : REAL := 0.0;
    op_trichain/outputChain/chain/m33 AT 352 : REAL := 100.0;
    op_trichain/outputChain/chain/m34 AT 353 : REAL := 1.06;
    op_trichain/outputChain/chain/m41 AT 354 : REAL := 0.0;
    op_trichain/outputChain/chain/m42 AT 355 : REAL := 0.0;
    op_trichain/outputChain/chain/m43 AT 356 : REAL := 0.0;
    op_trichain/outputChain/chain/m44 AT 357 : REAL := 1.0;
    op_trichain/outputChain/chain/px AT 358 : REAL := 7100.0;
    op_trichain/outputChain/chain/py AT 359 : REAL := 3000.0;
    op_trichain/outputChain/chain/pz AT 360 : REAL := 0.0;
    op_trichain/outputChain/chain/dx AT 361 : REAL := 4000.0;
    op_trichain/outputChain/chain/dy AT 362 : REAL := 10000.0;
    op_trichain/outputChain/chain/dz AT 363 : REAL := 100.0;
    op_trichain/outputChain/chain/sProduct AT 364 : REAL := 0.0;
    op_trichain/outputChain/chain/interaction AT 254 : BOOL := false;
    op_trichain/outputChain/chain/d_locking AT 255 : BOOL := false;
    op_trichain/outputChain/chain/v_d_locking AT 256 : BOOL := false;
    op_trichain/shuttle/forward AT 25 : BOOL := false;
    op_trichain/shuttle/backward AT 24 : BOOL := false;
    op_trichain/shuttle/chainMotorOn AT 26 : BOOL := false;
    op_trichain/shuttle/sensor_Pos1 AT 15 : BOOL := false;
    op_trichain/shuttle/sensor_Pos2 AT 16 : BOOL := false;
    op_trichain/shuttle/sensor_Pos3 AT 17 : BOOL := false;
    op_trichain/shuttle/end_sensor AT 18 : BOOL := false;
    op_trichain/shuttle/motor2dir/forward AT 25 : BOOL := false;
    op_trichain/shuttle/motor2dir/backward AT 24 : BOOL := false;
    op_trichain/shuttle/motor2dir/cmdSupply AT 271 : BOOL := true;
    op_trichain/shuttle/motor2dir/sensorSupply AT 270 : BOOL := true;
    op_trichain/shuttle/motor2dir/voltage380 AT 269 : BOOL := true;
    op_trichain/shuttle/motor2dir/speedVal AT 369 : REAL := 0.0;
    op_trichain/shuttle/motor2dir/speedPercent AT 368 : REAL := 0.0;
    op_trichain/shuttle/motor2dir/thermal AT 268 : BOOL := false;
    op_trichain/shuttle/motor2dir/backwardFB AT 267 : BOOL := false;
    op_trichain/shuttle/motor2dir/forwardFB AT 266 : BOOL := false;
    op_trichain/shuttle/motor2dir/increment AT 372 : REAL := 0.0;
    op_trichain/shuttle/motor2dir/memoFwd AT 272 : BOOL := false;
    op_trichain/shuttle/motor2dir/memoBwd AT 273 : BOOL := false;
    op_trichain/shuttle/motor2dir/forwardState AT 274 : BOOL := false;
    op_trichain/shuttle/motor2dir/backwardState AT 275 : BOOL := false;
    op_trichain/shuttle/motor2dir/wantedSpeed AT 373 : REAL := 0.0;
    op_trichain/shuttle/motor2dir/nominalSpeed AT 374 : REAL := 500.0;
    op_trichain/shuttle/motor2dir/nominalTime AT 375 : REAL := 0.1;
    op_trichain/shuttle/motor2dir/thermalLogic AT 276 : BOOL := false;
    op_trichain/shuttle/motor2dir/fwdFbLogic AT 277 : BOOL := true;
    op_trichain/shuttle/motor2dir/bwdFbLogic AT 278 : BOOL := true;
    op_trichain/shuttle/motor2dir/d_locking AT 279 : BOOL := false;
    op_trichain/shuttle/motor2dir/v_d_locking AT 376 : REAL := 0.0;
    op_trichain/shuttle/motor2dir/d_electrical AT 280 : BOOL := false;
    op_trichain/shuttle/motor2dir/v_d_electrical AT 281 : BOOL := false;
    op_trichain/shuttle/motor2dir/d_backwardFB AT 282 : BOOL := false;
    op_trichain/shuttle/motor2dir/v_d_backwardFB AT 283 : BOOL := false;
    op_trichain/shuttle/motor2dir/d_forwardFB AT 284 : BOOL := false;
    op_trichain/shuttle/motor2dir/v_d_forwardFB AT 285 : BOOL := false;
    op_trichain/shuttle/chainMotor/forward AT 26 : BOOL := false;
    op_trichain/shuttle/chainMotor/cmdSupply AT 265 : BOOL := true;
    op_trichain/shuttle/chainMotor/sensorSupply AT 264 : BOOL := true;
    op_trichain/shuttle/chainMotor/voltage380 AT 263 : BOOL := true;
    op_trichain/shuttle/chainMotor/speedVal AT 370 : REAL := 0.0;
    op_trichain/shuttle/chainMotor/speedPercent AT 367 : REAL := 0.0;
    op_trichain/shuttle/chainMotor/thermal AT 262 : BOOL := false;
    op_trichain/shuttle/chainMotor/forwardFB AT 261 : BOOL := false;
    op_trichain/shuttle/chainMotor/increment AT 377 : REAL := 0.0;
    op_trichain/shuttle/chainMotor/memoFwd AT 286 : BOOL := false;
    op_trichain/shuttle/chainMotor/forwardState AT 287 : BOOL := false;
    op_trichain/shuttle/chainMotor/wantedSpeed AT 378 : REAL := 0.0;
    op_trichain/shuttle/chainMotor/nominalSpeed AT 379 : REAL := 500.0;
    op_trichain/shuttle/chainMotor/nominalTime AT 380 : REAL := 0.1;
    op_trichain/shuttle/chainMotor/thermalLogic AT 288 : BOOL := false;
    op_trichain/shuttle/chainMotor/feedbackLogic AT 289 : BOOL := true;
    op_trichain/shuttle/chainMotor/d_locking AT 290 : BOOL := false;
    op_trichain/shuttle/chainMotor/v_d_locking AT 381 : REAL := 0.0;
    op_trichain/shuttle/chainMotor/d_feedback AT 291 : BOOL := false;
    op_trichain/shuttle/chainMotor/v_d_feedback AT 292 : BOOL := false;
    op_trichain/shuttle/chainMotor/d_electrical AT 293 : BOOL := false;
    op_trichain/shuttle/chainMotor/v_d_electrical AT 294 : BOOL := false;
    op_trichain/shuttle/axle/speed AT 369 : REAL := 0.0;
    op_trichain/shuttle/axle/positionTranslat AT 371 : REAL := 0.0;
    op_trichain/shuttle/axle/percentTranslat AT 366 : REAL := 0.0;
    op_trichain/shuttle/axle/incTranslat AT 365 : REAL := 0.0;
    op_trichain/shuttle/axle/firstCycle AT 295 : BOOL := false;
    op_trichain/shuttle/axle/nbCyclePerSec AT 382 : REAL := 0.0;
    op_trichain/shuttle/axle/initTranslat AT 383 : REAL := 5100.0;
    op_trichain/shuttle/axle/maxTranslat AT 384 : REAL := 30000.0;
    op_trichain/shuttle/axle/minTranslat AT 385 : REAL := 0.0;
    op_trichain/shuttle/axle/d_locking AT 296 : BOOL := false;
    op_trichain/shuttle/axle/v_d_locking AT 297 : BOOL := false;
    op_trichain/shuttle/shuttle/speedX AT 369 : REAL := 0.0;
    op_trichain/shuttle/shuttle/speedY AT 370 : REAL := 0.0;
    op_trichain/shuttle/shuttle/status_act_prod AT 540 : DINT := 0;
    op_trichain/shuttle/shuttle/m11 AT 386 : REAL := 2997.32;
    op_trichain/shuttle/shuttle/m12 AT 387 : REAL := 0.0;
    op_trichain/shuttle/shuttle/m13 AT 388 : REAL := -2.44921e-014;
    op_trichain/shuttle/shuttle/m14 AT 389 : REAL := 5231.25;
    op_trichain/shuttle/shuttle/m21 AT 390 : REAL := 0.0;
    op_trichain/shuttle/shuttle/m22 AT 391 : REAL := 7497.32;
    op_trichain/shuttle/shuttle/m23 AT 392 : REAL := 0.0;
    op_trichain/shuttle/shuttle/m24 AT 393 : REAL := 11601.8;
    op_trichain/shuttle/shuttle/m31 AT 394 : REAL := 7.34108e-013;
    op_trichain/shuttle/shuttle/m32 AT 395 : REAL := 0.0;
    op_trichain/shuttle/shuttle/m33 AT 396 : REAL := 100.0;
    op_trichain/shuttle/shuttle/m34 AT 397 : REAL := 1.05;
    op_trichain/shuttle/shuttle/m41 AT 398 : REAL := 0.0;
    op_trichain/shuttle/shuttle/m42 AT 399 : REAL := 0.0;
    op_trichain/shuttle/shuttle/m43 AT 400 : REAL := 0.0;
    op_trichain/shuttle/shuttle/m44 AT 401 : REAL := 1.0;
    op_trichain/shuttle/shuttle/px AT 402 : REAL := 5250.0;
    op_trichain/shuttle/shuttle/py AT 403 : REAL := 11600.0;
    op_trichain/shuttle/shuttle/pz AT 404 : REAL := 1.05;
    op_trichain/shuttle/shuttle/dx AT 405 : REAL := 3000.0;
    op_trichain/shuttle/shuttle/dy AT 406 : REAL := 7500.0;
    op_trichain/shuttle/shuttle/dz AT 407 : REAL := 100.0;
    op_trichain/shuttle/shuttle/sProdX AT 408 : REAL := 0.0;
    op_trichain/shuttle/shuttle/sProdY AT 409 : REAL := 0.0;
    op_trichain/shuttle/shuttle/d_locking AT 298 : BOOL := false;
    op_trichain/shuttle/shuttle/v_d_locking AT 299 : BOOL := false;
    op_trichain/shuttle/pos1Sensor/level AT 371 : REAL := 0.0;
    op_trichain/shuttle/pos1Sensor/sensorSupply AT 260 : BOOL := true;
    op_trichain/shuttle/pos1Sensor/rangeSensor AT 15 : BOOL := false;
    op_trichain/shuttle/pos1Sensor/status_act_prod AT 541 : DINT := 0;
    op_trichain/shuttle/pos1Sensor/m11 AT 410 : REAL := 498.214;
    op_trichain/shuttle/pos1Sensor/m12 AT 411 : REAL := 0.0;
    op_trichain/shuttle/pos1Sensor/m13 AT 412 : REAL := 0.0;
    op_trichain/shuttle/pos1Sensor/m14 AT 413 : REAL := 3479.47;
    op_trichain/shuttle/pos1Sensor/m21 AT 414 : REAL := 0.0;
    op_trichain/shuttle/pos1Sensor/m22 AT 415 : REAL := 498.214;
    op_trichain/shuttle/pos1Sensor/m23 AT 416 : REAL := 0.0;
    op_trichain/shuttle/pos1Sensor/m24 AT 417 : REAL := 17998.2;
    op_trichain/shuttle/pos1Sensor/m31 AT 418 : REAL := 0.0;
    op_trichain/shuttle/pos1Sensor/m32 AT 419 : REAL := 0.0;
    op_trichain/shuttle/pos1Sensor/m33 AT 420 : REAL := 100.0;
    op_trichain/shuttle/pos1Sensor/m34 AT 421 : REAL := 1.05;
    op_trichain/shuttle/pos1Sensor/m41 AT 422 : REAL := 0.0;
    op_trichain/shuttle/pos1Sensor/m42 AT 423 : REAL := 0.0;
    op_trichain/shuttle/pos1Sensor/m43 AT 424 : REAL := 0.0;
    op_trichain/shuttle/pos1Sensor/m44 AT 425 : REAL := 1.0;
    op_trichain/shuttle/pos1Sensor/threshold AT 426 : REAL := 900.0;
    op_trichain/shuttle/pos1Sensor/range AT 427 : REAL := 900.0;
    op_trichain/shuttle/pos1Sensor/wiringLogic AT 300 : BOOL := true;
    op_trichain/shuttle/pos1Sensor/d_sensor AT 301 : BOOL := false;
    op_trichain/shuttle/pos1Sensor/v_d_sensor AT 302 : BOOL := false;
    op_trichain/shuttle/pos2Sensor/level AT 371 : REAL := 0.0;
    op_trichain/shuttle/pos2Sensor/sensorSupply AT 259 : BOOL := true;
    op_trichain/shuttle/pos2Sensor/rangeSensor AT 16 : BOOL := false;
    op_trichain/shuttle/pos2Sensor/status_act_prod AT 542 : DINT := 0;
    op_trichain/shuttle/pos2Sensor/m11 AT 428 : REAL := 500.0;
    op_trichain/shuttle/pos2Sensor/m12 AT 429 : REAL := 0.0;
    op_trichain/shuttle/pos2Sensor/m13 AT 430 : REAL := 0.0;
    op_trichain/shuttle/pos2Sensor/m14 AT 431 : REAL := 7000.0;
    op_trichain/shuttle/pos2Sensor/m21 AT 432 : REAL := 0.0;
    op_trichain/shuttle/pos2Sensor/m22 AT 433 : REAL := 500.0;
    op_trichain/shuttle/pos2Sensor/m23 AT 434 : REAL := 0.0;
    op_trichain/shuttle/pos2Sensor/m24 AT 435 : REAL := 18000.0;
    op_trichain/shuttle/pos2Sensor/m31 AT 436 : REAL := 0.0;
    op_trichain/shuttle/pos2Sensor/m32 AT 437 : REAL := 0.0;
    op_trichain/shuttle/pos2Sensor/m33 AT 438 : REAL := 100.0;
    op_trichain/shuttle/pos2Sensor/m34 AT 439 : REAL := 1.06;
    op_trichain/shuttle/pos2Sensor/m41 AT 440 : REAL := 0.0;
    op_trichain/shuttle/pos2Sensor/m42 AT 441 : REAL := 0.0;
    op_trichain/shuttle/pos2Sensor/m43 AT 442 : REAL := 0.0;
    op_trichain/shuttle/pos2Sensor/m44 AT 443 : REAL := 1.0;
    op_trichain/shuttle/pos2Sensor/threshold AT 444 : REAL := 4500.0;
    op_trichain/shuttle/pos2Sensor/range AT 445 : REAL := 900.0;
    op_trichain/shuttle/pos2Sensor/wiringLogic AT 303 : BOOL := true;
    op_trichain/shuttle/pos2Sensor/d_sensor AT 304 : BOOL := false;
    op_trichain/shuttle/pos2Sensor/v_d_sensor AT 305 : BOOL := false;
    op_trichain/shuttle/pos3Sensor/level AT 371 : REAL := 0.0;
    op_trichain/shuttle/pos3Sensor/sensorSupply AT 258 : BOOL := true;
    op_trichain/shuttle/pos3Sensor/rangeSensor AT 17 : BOOL := false;
    op_trichain/shuttle/pos3Sensor/status_act_prod AT 543 : DINT := 0;
    op_trichain/shuttle/pos3Sensor/m11 AT 446 : REAL := 500.0;
    op_trichain/shuttle/pos3Sensor/m12 AT 447 : REAL := 0.0;
    op_trichain/shuttle/pos3Sensor/m13 AT 448 : REAL := 0.0;
    op_trichain/shuttle/pos3Sensor/m14 AT 449 : REAL := 11400.0;
    op_trichain/shuttle/pos3Sensor/m21 AT 450 : REAL := 0.0;
    op_trichain/shuttle/pos3Sensor/m22 AT 451 : REAL := 500.0;
    op_trichain/shuttle/pos3Sensor/m23 AT 452 : REAL := 0.0;
    op_trichain/shuttle/pos3Sensor/m24 AT 453 : REAL := 18000.0;
    op_trichain/shuttle/pos3Sensor/m31 AT 454 : REAL := 0.0;
    op_trichain/shuttle/pos3Sensor/m32 AT 455 : REAL := 0.0;
    op_trichain/shuttle/pos3Sensor/m33 AT 456 : REAL := 100.0;
    op_trichain/shuttle/pos3Sensor/m34 AT 457 : REAL := 0.0;
    op_trichain/shuttle/pos3Sensor/m41 AT 458 : REAL := 0.0;
    op_trichain/shuttle/pos3Sensor/m42 AT 459 : REAL := 0.0;
    op_trichain/shuttle/pos3Sensor/m43 AT 460 : REAL := 0.0;
    op_trichain/shuttle/pos3Sensor/m44 AT 461 : REAL := 1.0;
    op_trichain/shuttle/pos3Sensor/threshold AT 462 : REAL := 9200.0;
    op_trichain/shuttle/pos3Sensor/range AT 463 : REAL := 900.0;
    op_trichain/shuttle/pos3Sensor/wiringLogic AT 306 : BOOL := true;
    op_trichain/shuttle/pos3Sensor/d_sensor AT 307 : BOOL := false;
    op_trichain/shuttle/pos3Sensor/v_d_sensor AT 308 : BOOL := false;
    op_trichain/shuttle/endSensor/sensorSupply AT 257 : BOOL := true;
    op_trichain/shuttle/endSensor/deltaTranslation AT 371 : REAL := 0.0;
    op_trichain/shuttle/endSensor/passing AT 18 : BOOL := false;
    op_trichain/shuttle/endSensor/status_act_prod AT 544 : DINT := 0;
    op_trichain/shuttle/endSensor/m11 AT 464 : REAL := 337.5;
    op_trichain/shuttle/endSensor/m12 AT 465 : REAL := 0.0;
    op_trichain/shuttle/endSensor/m13 AT 466 : REAL := 0.0;
    op_trichain/shuttle/endSensor/m14 AT 467 : REAL := 5464.29;
    op_trichain/shuttle/endSensor/m21 AT 468 : REAL := 0.0;
    op_trichain/shuttle/endSensor/m22 AT 469 : REAL := 369.643;
    op_trichain/shuttle/endSensor/m23 AT 470 : REAL := 0.0;
    op_trichain/shuttle/endSensor/m24 AT 471 : REAL := 13032.1;
    op_trichain/shuttle/endSensor/m31 AT 472 : REAL := 0.0;
    op_trichain/shuttle/endSensor/m32 AT 473 : REAL := 0.0;
    op_trichain/shuttle/endSensor/m33 AT 474 : REAL := 100.0;
    op_trichain/shuttle/endSensor/m34 AT 475 : REAL := 1.0;
    op_trichain/shuttle/endSensor/m41 AT 476 : REAL := 0.0;
    op_trichain/shuttle/endSensor/m42 AT 477 : REAL := 0.0;
    op_trichain/shuttle/endSensor/m43 AT 478 : REAL := 0.0;
    op_trichain/shuttle/endSensor/m44 AT 479 : REAL := 1.0;
    op_trichain/shuttle/endSensor/px AT 480 : REAL := 0.0;
    op_trichain/shuttle/endSensor/py AT 481 : REAL := 14500.0;
    op_trichain/shuttle/endSensor/pz AT 482 : REAL := 0.0;
    op_trichain/shuttle/endSensor/dx AT 483 : REAL := 500.0;
    op_trichain/shuttle/endSensor/dy AT 484 : REAL := 500.0;
    op_trichain/shuttle/endSensor/dz AT 485 : REAL := 100.0;
    op_trichain/shuttle/endSensor/detection AT 309 : BOOL := false;
    op_trichain/shuttle/endSensor/passingLogic AT 310 : BOOL := true;
    op_trichain/shuttle/endSensor/initialPosition AT 486 : REAL := 1000.0;
    op_trichain/shuttle/endSensor/d_passing AT 311 : BOOL := false;
    op_trichain/shuttle/endSensor/v_d_passing AT 312 : BOOL := false;
    op_trichain/runButton/output AT 5 : BOOL := false;
    op_trichain/runButton/user_PushButton AT 313 : BOOL := false;
    op_trichain/runButton/time2reach AT 314 : BOOL := false;
    op_trichain/runButton/pulse_type AT 315 : BOOL := false;
    op_trichain/runButton/pulseDuration AT 487 : REAL := 2.0;
    op_trichain/creation3/idProd AT 523 : DINT := 0;
    op_trichain/creation3/creationFailed AT 122 : BOOL := false;
    op_trichain/creation3/status_act_prod AT 545 : DINT := 0;
    op_trichain/creation3/m11 AT 488 : REAL := 1500.0;
    op_trichain/creation3/m12 AT 489 : REAL := 0.0;
    op_trichain/creation3/m13 AT 490 : REAL := 0.0;
    op_trichain/creation3/m14 AT 491 : REAL := 13000.0;
    op_trichain/creation3/m21 AT 492 : REAL := 0.0;
    op_trichain/creation3/m22 AT 493 : REAL := 3000.0;
    op_trichain/creation3/m23 AT 494 : REAL := 0.0;
    op_trichain/creation3/m24 AT 495 : REAL := 27000.0;
    op_trichain/creation3/m31 AT 496 : REAL := 0.0;
    op_trichain/creation3/m32 AT 497 : REAL := 0.0;
    op_trichain/creation3/m33 AT 498 : REAL := 100.0;
    op_trichain/creation3/m34 AT 499 : REAL := 0.0;
    op_trichain/creation3/m41 AT 500 : REAL := 0.0;
    op_trichain/creation3/m42 AT 501 : REAL := 0.0;
    op_trichain/creation3/m43 AT 502 : REAL := 0.0;
    op_trichain/creation3/m44 AT 503 : REAL := 1.0;
    op_trichain/creation3/px AT 504 : REAL := 12990.0;
    op_trichain/creation3/py AT 505 : REAL := 27000.0;
    op_trichain/creation3/pz AT 506 : REAL := 1.5;
    op_trichain/creation3/dx AT 507 : REAL := 1500.0;
    op_trichain/creation3/dy AT 508 : REAL := 3000.0;
    op_trichain/creation3/dz AT 509 : REAL := 100.0;
    op_trichain/creation3/presenceProduct AT 316 : BOOL := false;
    op_trichain/creation3/arrival_PB AT 317 : BOOL := false;
    op_trichain/creation3/time2reach AT 510 : REAL := 0.0;
    op_trichain/creation3/edge_arrival_PB AT 318 : BOOL := false;
    op_trichain/creation3/first AT 319 : BOOL := true;
    op_trichain/creation3/pulseType AT 320 : BOOL := true;
    op_trichain/creation3/pulseDuration AT 511 : REAL := 10.0;
    op_trichain/trash/status_act_prod AT 546 : DINT := 0;
    op_trichain/trash/m11 AT 512 : REAL := 1197.32;
    op_trichain/trash/m12 AT 513 : REAL := 0.0;
    op_trichain/trash/m13 AT 514 : REAL := -2.44921e-014;
    op_trichain/trash/m14 AT 515 : REAL := 7103.57;
    op_trichain/trash/m21 AT 516 : REAL := 0.0;
    op_trichain/trash/m22 AT 517 : REAL := 2499.11;
    op_trichain/trash/m23 AT 518 : REAL := 0.0;
    op_trichain/trash/m24 AT 519 : REAL := 841.954;
    op_trichain/trash/m31 AT 520 : REAL := 2.9325e-013;
    op_trichain/trash/m32 AT 521 : REAL := 0.0;
    op_trichain/trash/m33 AT 522 : REAL := 100.0;
    op_trichain/trash/m34 AT 523 : REAL := 1.0;
    op_trichain/trash/m41 AT 524 : REAL := 0.0;
    op_trichain/trash/m42 AT 525 : REAL := 0.0;
    op_trichain/trash/m43 AT 526 : REAL := 0.0;
    op_trichain/trash/m44 AT 527 : REAL := 1.0;
    op_trichain/trash/px AT 528 : REAL := 7100.0;
    op_trichain/trash/py AT 529 : REAL := 1400.0;
    op_trichain/trash/pz AT 530 : REAL := 0.0;
    op_trichain/trash/dx AT 531 : REAL := 1200.0;
    op_trichain/trash/dy AT 532 : REAL := 2500.0;
    op_trichain/trash/dz AT 533 : REAL := 100.0;
  END_VAR
END_CONFIGURATION
